// TIA Portal V20 export
// export: Created 2026-07-14T21:06:33.1463258Z, ExportSetting WithDefaults, DisplayName Totally Integrated Automation Portal, DisplayVersion V20 Update 5, DisplayName TIA Portal Openness, DisplayVersion V20 Update 4, DisplayName TIA Portal Version Control Interface, DisplayVersion V20 Update 5, DisplayName SINAMICS Startdrive Advanced, DisplayVersion V20, DisplayName SINAMICS DCC, DisplayVersion V20, DisplayName SINAMICS Startdrive G130, G150, S120, S150, SINAMICS MV, G220, S200, S210, DisplayVersion V20, DisplayName SINAMICS Startdrive G110M, G120, G120C, G120D, G120P, G115D, DisplayVersion V20, DisplayName STEP 7 Professional, DisplayVersion V20 Update 5, DisplayName STEP 7 Safety, DisplayVersion V20 Update 2, DisplayName WinCC Basic/Comfort/Advanced, DisplayVersion V20 Update 5, DisplayName WinCC Unified, DisplayVersion V20 Update 5
FUNCTION "TimerSample" : Void   // FC1, LAD
TITLE = Chained On-Delay Timer Sequence
{ S7_Optimized_Access := 'TRUE' }
VERSION : 0.1
// stored: AutoNumber true, IsIECCheckEnabled false, SetENOAutomatically false, UDAEnableTagReadback false
BEGIN

REGION Network 1: Timer 0: Fixed 100ms Preset
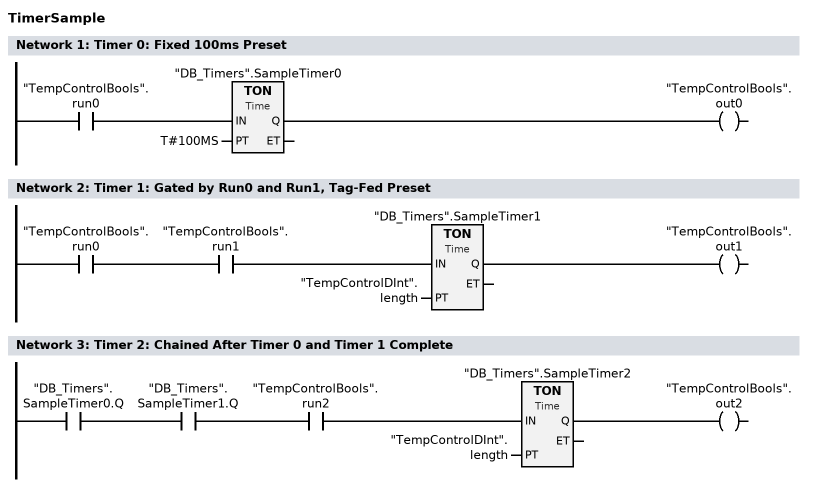
   RUNG wire#powerrail
      Contact( "TempControlBools".run0 )
      { S7_Templates := "time_type := Time" } "DB_Timers".SampleTimer0.TON(pt := T#100MS, et =>)
      Coil( "TempControlBools".out0 )
   END_RUNG
   // the same network as SCL:
   "DB_Timers".SampleTimer0.TON(IN := "TempControlBools".run0, PT := T#100MS);
   "TempControlBools".out0 := "DB_Timers".SampleTimer0.Q;
END_REGION

REGION Network 2: Timer 1: Gated by Run0 and Run1, Tag-Fed Preset
   RUNG wire#powerrail
      Contact( "TempControlBools".run0 )
      Contact( "TempControlBools".run1 )
      { S7_Templates := "time_type := Time" } "DB_Timers".SampleTimer1.TON(pt := "TempControlDInt".length, et =>)
      Coil( "TempControlBools".out1 )
   END_RUNG
   // the same network as SCL:
   "DB_Timers".SampleTimer1.TON(IN := "TempControlBools".run0 AND "TempControlBools".run1,
                           PT := "TempControlDInt".length);
   "TempControlBools".out1 := "DB_Timers".SampleTimer1.Q;
END_REGION

REGION Network 3: Timer 2: Chained After Timer 0 and Timer 1 Complete
   RUNG wire#powerrail
      Contact( "DB_Timers".SampleTimer0.Q )
      Contact( "DB_Timers".SampleTimer1.Q )
      Contact( "TempControlBools".run2 )
      { S7_Templates := "time_type := Time" } "DB_Timers".SampleTimer2.TON(pt := "TempControlDInt".length, et =>)
      Coil( "TempControlBools".out2 )
   END_RUNG
   // the same network as SCL:
   "DB_Timers".SampleTimer2.TON(IN := "DB_Timers".SampleTimer0.Q AND "DB_Timers".SampleTimer1.Q AND "TempControlBools".run2,
                           PT := "TempControlDInt".length);
   "TempControlBools".out2 := "DB_Timers".SampleTimer2.Q;
END_REGION
END_FUNCTION
